VAR_GLOBAL
	stPlantConfiguration	: ST_PlantConfiguration;
	wsJson					: WSTRING(20000);
END_VAR

(* stored: Version 1.1.0.1, ProductVersion 3.1.4024.4
   GVL ReactorManager: Id {685bfe84-bef6-45a6-bd0b-f7d743fa3d30} *)
